(* IEC 61131-3 sources: Lasal/CPU_5344_V01/Class/Bridge, 1 file *)

(* ---- Bridge.st ---- *)
(*!
<Class
	Name               = "Bridge"
	Revision           = "1.0"
	RealtimeTask       = "false"
	CyclicTask         = "true"
	BackgroundTask     = "false"
	Sigmatek           = "true"
	OSInterface        = "false"
	HighPriority       = "false"
	Automatic          = "false"
	UpdateMode         = "Prescan"
	IconPath           = ".\Class\Bridge\bridge.ico"
	SharedCommandTable = "true"
	Objectsize         = "(284,120)"
	Comment            = "V1.0&#13;&#10;Claas reads the first Client &#13;&#10;and writes the value on the next.&#13;&#10;To use it turn on the cyclic time">
	<Channels>
		<Server Name="dummy" Visualized="true" Initialize="false" WriteProtected="false" Retentive="false" Comment="no use"/>
		<Client Name="Client_Read" Required="false" Internal="false" Comment="reading Client"/>
		<Client Name="Client_Write" Required="false" Internal="false" Comment="Client_Write = Client_Read"/>
	</Channels>
</Class>
*)
Bridge : CLASS
  //Servers:
	dummy 	: SvrChCmd_DINT;
  //Clients:
	Client_Read 	: CltCh_DINT;
	Client_Write 	: CltCh_DINT;
  //Variables:
  //Functions:
				//! <Function Comment=" ******************************************************************&#13;&#10;   Klasse liest den ersten Client und schreibt den zweiten Client&#13;&#10; ******************************************************************&#13;&#10;    erstellt    :   BS  :     KW 35/01&#13;&#10; ******************************************************************&#13;&#10;                           CYWORK Funktion&#13;&#10; ******************************************************************&#13;&#10;   getested: BS | 29.11.2001 | Lasal V00.53 | OPS V4.00&#13;&#10; ******************************************************************&#13;&#10; ******************************************************************&#13;&#10;            Class reads the first Client and writes the&#13;&#10;                          next Client&#13;&#10; ******************************************************************&#13;&#10;    created    :   BS  :     KW 35/01&#13;&#10; ******************************************************************&#13;&#10;                    Operation of CyWork Function&#13;&#10; ******************************************************************&#13;&#10;   tested: BS | 29.11.2001 | Lasal V00.53 | OPS V4.00&#13;&#10; ******************************************************************&#13;&#10;" Name="CyWork"/>
	FUNCTION VIRTUAL GLOBAL CyWork
		VAR_INPUT
			EAX 	: UDINT := EAX;
		END_VAR
		VAR_OUTPUT
			state (EAX) 	: UDINT;
		END_VAR;
  //Tables:
	FUNCTION @STD
		VAR_OUTPUT
			ret_code	: CONFSTATES;
		END_VAR;
	FUNCTION GLOBAL TAB @CT_;
END_CLASS;

//*********************Inserted from .\code\C_Bridge.st*********************

//[#DEUTSCH]
// ******************************************************************
//   Klasse liest den ersten Client und schreibt den zweiten Client
// ******************************************************************
//  		erstellt 		 :		 BS		:   		KW 35/01
// ******************************************************************
//                           CYWORK Funktion
// ******************************************************************
//   getested: BS | 29.11.2001 | Lasal V00.53 | OPS V4.00
// ******************************************************************
//[#ENGLISH]
// ******************************************************************
//            Class reads the first Client and writes the
//                          next Client
// ******************************************************************
//  		created 		 :		 BS		:   		KW 35/01
// ******************************************************************
//                    Operation of CyWork Function
// ******************************************************************
//   tested: BS | 29.11.2001 | Lasal V00.53 | OPS V4.00
// ******************************************************************
FUNCTION VIRTUAL GLOBAL Bridge::CyWork
VAR_INPUT
	EAX		: UDINT;
END_VAR
VAR_OUTPUT
	state		: UDINT;
END_VAR

	Client_Read	:= Client_Read.Read();
	Client_Write:= Client_Read;
	Client_Write.Write(Client_Write);

	state := READY$UDINT;
END_FUNCTION //VIRTUAL GLOBAL Bridge::CyWork
